% RSLogix 500 project PACKAGING_BAK001.RSS, saved by version 8.30.00.16 %
PROJECT "UNTITLED"    % processor: MicroLogix 1000 %

PROGRAM FILES
  LAD 2 "MAIN_PROG"  23 rungs
  LAD 3 "USER_FAULT"  1 rungs
  LAD 4 "HSC_INT"  1 rungs
  LAD 5 "STI_INT"  1 rungs
  LAD 6, 7, 8, 9, 10, 11, 12, 13, 14, 15, 16: only END

DATA FILES
  O0 OUTPUT  1 elements
  I1 INPUT  2 elements
  S2 STATUS  33 elements
  B3 BINARY  32 elements
  T4 TIMER  40 elements
  C5 COUNTER  32 elements
  R6 CONTROL  16 elements
  N7 INTEGER  105 elements

LADDER 2 "MAIN_PROG"
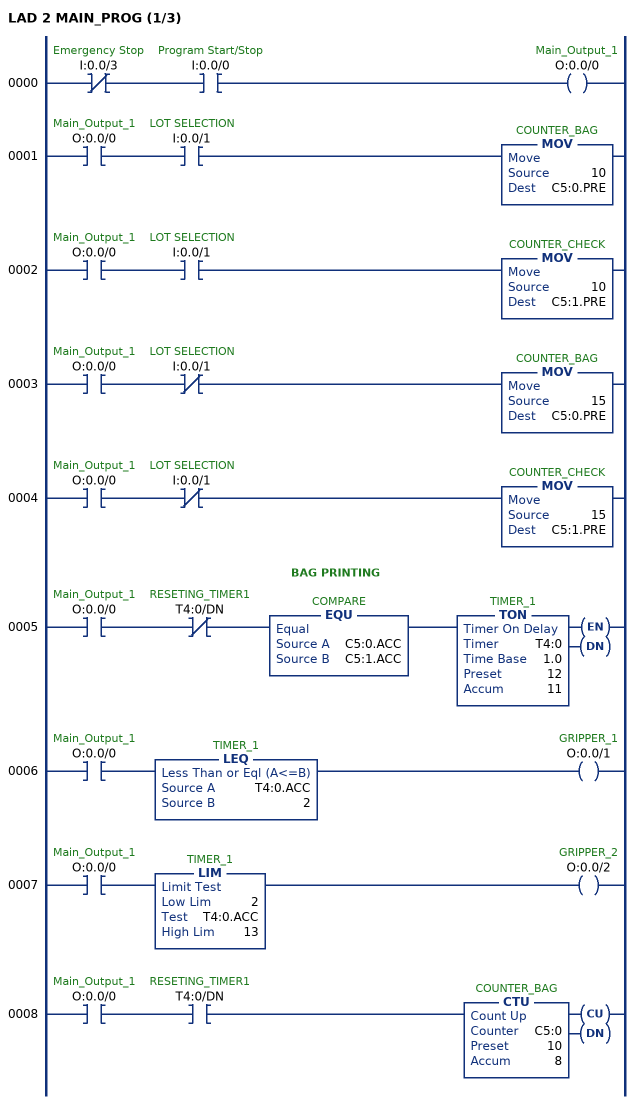
% Rung: 0 %
SOR XIO I:0.0/3 XIC I:0.0/0 OTE O:0.0/0 EOR
%   I:0.0/3  "Emergency Stop" %
%   I:0.0/0  "Program Start/Stop" %
%   O:0.0/0  "Main_Output_1" %
% Rung: 1 %
SOR XIC O:0.0/0 XIC I:0.0/1 MOV 10 C5:0.PRE EOR
%   O:0.0/0  "Main_Output_1" %
%   I:0.0/1  "LOT SELECTION" %
%   C5:0  "COUNTER_BAG" %
% Rung: 2 %
SOR XIC O:0.0/0 XIC I:0.0/1 MOV 10 C5:1.PRE EOR
%   O:0.0/0  "Main_Output_1" %
%   I:0.0/1  "LOT SELECTION" %
%   C5:1.PRE  "COUNTER_CHECK" %
% Rung: 3 %
SOR XIC O:0.0/0 XIO I:0.0/1 MOV 15 C5:0.PRE EOR
%   O:0.0/0  "Main_Output_1" %
%   I:0.0/1  "LOT SELECTION" %
%   C5:0  "COUNTER_BAG" %
% Rung: 4 %
SOR XIC O:0.0/0 XIO I:0.0/1 MOV 15 C5:1.PRE EOR
%   O:0.0/0  "Main_Output_1" %
%   I:0.0/1  "LOT SELECTION" %
%   C5:1.PRE  "COUNTER_CHECK" %
% Rung: 5 %
% TITLE: BAG PRINTING %
SOR XIC O:0.0/0 XIO T4:0/DN EQU C5:0.ACC C5:1.ACC TON T4:0 1.0 12 11 EOR
%   O:0.0/0  "Main_Output_1" %
%   T4:0/DN  "RESETING_TIMER1" %
%   C5:0.ACC  "COMPARE" %
%   C5:1.ACC  "COMPARE" %
%   T4:0  "TIMER_1" %
% Rung: 6 %
SOR XIC O:0.0/0 LEQ T4:0.ACC 2 OTE O:0.0/1 EOR
%   O:0.0/0  "Main_Output_1" %
%   T4:0  "TIMER_1" %
%   O:0.0/1  "GRIPPER_1" %
% Rung: 7 %
SOR XIC O:0.0/0 LIM 2 T4:0.ACC 13 OTE O:0.0/2 EOR
%   O:0.0/0  "Main_Output_1" %
%   T4:0  "TIMER_1" %
%   O:0.0/2  "GRIPPER_2" %
% Rung: 8 %
SOR XIC O:0.0/0 XIC T4:0/DN CTU C5:0 10 8 EOR
%   O:0.0/0  "Main_Output_1" %
%   T4:0/DN  "RESETING_TIMER1" %
%   C5:0  "COUNTER_BAG" %

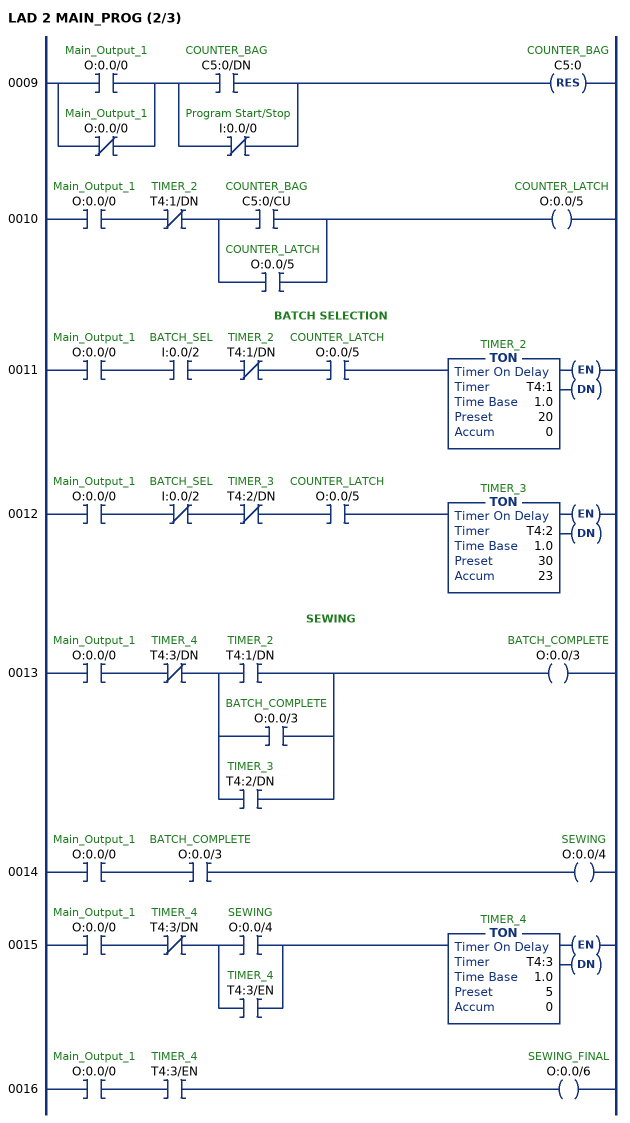
% Rung: 9 %
SOR BST XIC O:0.0/0 NXB XIO O:0.0/0 BND BST XIC C5:0/DN NXB XIO I:0.0/0 BND RES C5:0 EOR
%   O:0.0/0  "Main_Output_1" %
%   C5:0  "COUNTER_BAG" %
%   I:0.0/0  "Program Start/Stop" %
% Rung: 10 %
SOR XIC O:0.0/0 XIO T4:1/DN BST XIC C5:0/CU NXB XIC O:0.0/5 BND OTE O:0.0/5 EOR
%   O:0.0/0  "Main_Output_1" %
%   T4:1  "TIMER_2" %
%   C5:0  "COUNTER_BAG" %
%   O:0.0/5  "COUNTER_LATCH" %
% Rung: 11 %
% TITLE: BATCH SELECTION %
SOR XIC O:0.0/0 XIC I:0.0/2 XIO T4:1/DN XIC O:0.0/5 TON T4:1 1.0 20 0 EOR
%   O:0.0/0  "Main_Output_1" %
%   I:0.0/2  "BATCH_SEL" %
%   T4:1  "TIMER_2" %
%   O:0.0/5  "COUNTER_LATCH" %
% Rung: 12 %
SOR XIC O:0.0/0 XIO I:0.0/2 XIO T4:2/DN XIC O:0.0/5 TON T4:2 1.0 30 23 EOR
%   O:0.0/0  "Main_Output_1" %
%   I:0.0/2  "BATCH_SEL" %
%   T4:2  "TIMER_3" %
%   O:0.0/5  "COUNTER_LATCH" %
% Rung: 13 %
% TITLE: SEWING %
SOR XIC O:0.0/0 XIO T4:3/DN BST XIC T4:1/DN NXB XIC O:0.0/3 NXB XIC T4:2/DN BND OTE O:0.0/3 EOR
%   O:0.0/0  "Main_Output_1" %
%   T4:3  "TIMER_4" %
%   T4:1  "TIMER_2" %
%   O:0.0/3  "BATCH_COMPLETE" %
%   T4:2  "TIMER_3" %
% Rung: 14 %
SOR XIC O:0.0/0 XIC O:0.0/3 OTE O:0.0/4 EOR
%   O:0.0/0  "Main_Output_1" %
%   O:0.0/3  "BATCH_COMPLETE" %
%   O:0.0/4  "SEWING" %
% Rung: 15 %
SOR XIC O:0.0/0 XIO T4:3/DN BST XIC O:0.0/4 NXB XIC T4:3/EN BND TON T4:3 1.0 5 0 EOR
%   O:0.0/0  "Main_Output_1" %
%   T4:3  "TIMER_4" %
%   O:0.0/4  "SEWING" %
% Rung: 16 %
SOR XIC O:0.0/0 XIC T4:3/EN OTE O:0.0/6 EOR
%   O:0.0/0  "Main_Output_1" %
%   T4:3  "TIMER_4" %
%   O:0.0/6  "SEWING_FINAL" %

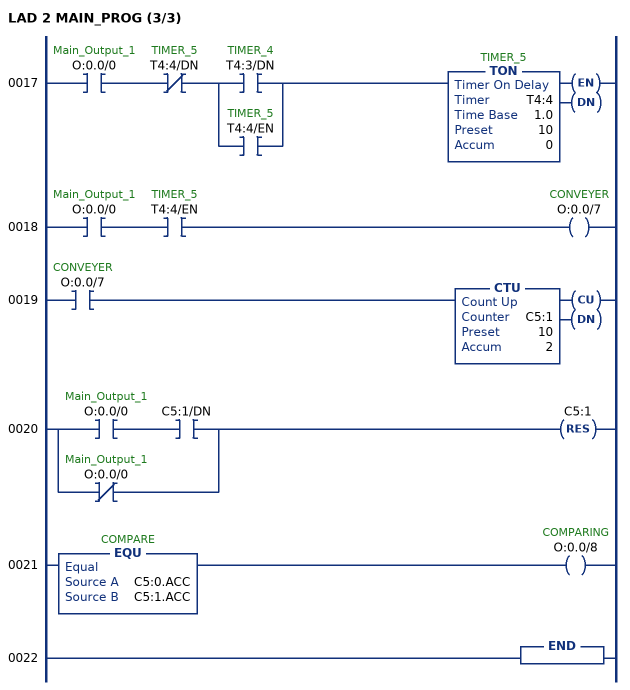
% Rung: 17 %
SOR XIC O:0.0/0 XIO T4:4/DN BST XIC T4:3/DN NXB XIC T4:4/EN BND TON T4:4 1.0 10 0 EOR
%   O:0.0/0  "Main_Output_1" %
%   T4:4  "TIMER_5" %
%   T4:3  "TIMER_4" %
% Rung: 18 %
SOR XIC O:0.0/0 XIC T4:4/EN OTE O:0.0/7 EOR
%   O:0.0/0  "Main_Output_1" %
%   T4:4  "TIMER_5" %
%   O:0.0/7  "CONVEYER" %
% Rung: 19 %
SOR XIC O:0.0/7 CTU C5:1 10 2 EOR
%   O:0.0/7  "CONVEYER" %
% Rung: 20 %
SOR BST XIC O:0.0/0 XIC C5:1/DN NXB XIO O:0.0/0 BND RES C5:1 EOR
%   O:0.0/0  "Main_Output_1" %
% Rung: 21 %
SOR EQU C5:0.ACC C5:1.ACC OTE O:0.0/8 EOR
%   C5:0.ACC  "COMPARE" %
%   C5:1.ACC  "COMPARE" %
%   O:0.0/8  "COMPARING" %
% Rung: 22 %
SOR END EOR

DATA TABLE (non-zero values as saved)
DATA T4
% .PRE .ACC %
% T4:0 % 12 11
% T4:1 % 20 0
% T4:2 % 30 23
% T4:3 % 5 0
% T4:4 % 10 0
DATA C5
% .PRE .ACC %
% C5:0 % 10 8
% C5:1 % 10 2
DATA N7
% N7:0 % 80 0 0 0 0 0 0 0 0 0
